//Manage data for read-only in PLC
stRoomDataPLC.bPirActive			:= stPirSensorData.bPrc;
stRoomDataPLC.uiActLuxLevel			:= TO_UINT(TRUNC(stPirSensorData.fBrightness));
stRoomDataPLC.uiActLightLevelPct	:= TO_UINT(TRUNC(arrfbLysGruppe[1].fbBallast.fActlLgtLvl_Prim));
		//stRoomDataPLC.uiActLightLevelPct	:= TO_UINT(TRUNC(fbLys.fbBallast.fActlLgtLvl_Prim)); //if only one group light control
stRoomDataPLC.uiBallastOnHours		:= uiBallastOnHours_MB; //The calculation for BallastOnHours is stored directly to the MB register below


//Assign data for read-only to MB registers
bPirActive_MB		:= stRoomDataPLC.bPirActive;
uiActLuxLevel_MB	:= stRoomDataPLC.uiActLuxLevel;

	//calculate BallastOnHours
	fbBallastOnHours(
		bEnableHourCount	:= bEnableHourCount,
		bPauseCount			:= arrfbLysGruppe[1].fbLightCtrl.bOffZone1,
		uiOnHours			:= uiBallastOnHours_MB,			//OnHours is updated here
		byOverflowCount		:= byOnHoursOverflowCount);


//Manage data for read/write for both PLC and MB registers
fbWriteSPLuxLevel(	nMaxValOut	:= uiMaxLuxLevel,
					nValIn1		:= uiSPLuxLevel_MB,		//nValIn1 takes priotity in case of download or restart
					nValIn2		:= stRoomDataPLC.uiSpLuxLevel,
					nValOut		=> uiLuxOn
				);


fbWritePirDelayTIme(	nMaxValOut	:= uiMaxPirOffMinutes,
						nValIn1		:= uiPirOffDelayTime_MB,		//nValIn1 takes priotity in case of download or restart
						nValIn2		:= stRoomDataPLC.uiPirOffDelayTime,
						nValOut		=> uiPirOffMinutes
					);
					

//Convert read/write modbus data to appropriate datatypes in PLC
fLuxOn	:= TO_REAL(uiLuxOn);			
tPIROff	:= TO_TIME(uiPirOffMinutes*udTimeScaling); //Time conversion defaults to ms

fLuxDim	:= TO_REAL(stRoomDataPLC.uiSpDimLuxLevel);			
tPIRDim	:= TO_TIME(stRoomDataPLC.uiPirDimDelayTime*udTimeScaling); //Time conversion defaults to ms
END_ACTION

ACTION A_Sensor:

fbSensor.ipCommunication := P_DALI_Background.arrfbKL6821Communication[Sensor_DALI_LINE_NUM];

//only 1 sensor
	
(*
fbSensor(
	byShrtAdr:= bySensorAddr,
	bInitialize:= bInitialize, 
	DALI_LINE_NUM:= Sensor_DALI_LINE_NUM, 
 	//bCancelHoldTimerOccupancy:= bCancelHoldTimerOccupancy, 
	stSensorSetup := stDaliSensorSetup,
	bInitErr=> bInitErr, 
	bInitDone=> bInitDone,
	stPirSensorData:= stPirSensorData, 
	arrSensorScales:= arrSensorScales);

*)
//several sensors	
fbSensor(
	arrShrtAdr:= arrSensorAddr,
	bInitialize:= bInitialize, 
	DALI_LINE_NUM:= Sensor_DALI_LINE_NUM, 
 	//bCancelHoldTimerOccupancy:= bCancelHoldTimerOccupancy, 
	stSensorSetup := stDaliSensorSetup,
	arrInitErr=> arrInitErr, 
	arrInitDone=> arrInitDone,
	stPirSensorData:= P_Foldedoer_4_517_Og_4_521_2Pcs.arrstPirSensorData_SepRoom[1], 
	arrSensorScales:= arrSensorScales);
	
	stPirSensorData := P_Foldedoer_4_517_Og_4_521_2Pcs.arrstPirSensorData_SepRoom[1]; //For at holde navngivning i ModbusComm
END_ACTION

END_PROGRAM

// ---- POUs/Alle_Rum/Rum_Med_DALI_Pir/Rum_4_513_Og_4_517_Og_4_521_Foldedoer/P_Rum_4_517.TcPOU
PROGRAM P_Rum_4_517
VAR

	arrfbLysGruppe			: ARRAY [1..2] OF FB_Light_Type_A;
	arrstDaliSetupGruppe	: ARRAY[1..2] OF SH_Light.ST_DALI_RoomSetup := 
	
													[(	byShrtAdr_Prim := 32, 
														byGrpAdr_Prim := 5, 
														eMod_Prim := E_DALIAddressType.Group, 
														//byShrtAdr_Sec := 1, 
														//byGrpAdr_Sec := 1, 
														//eMod_Sec := E_DALIAddressType.Short, 
														//byShrtAdr_Supl := 1,
														//eMod_Supl := E_DALIADDRESSTYPE.Group,
                                                        //byGrpAdr_Supl := 0, 
														DALI_LINE_NUM_PRIM := arrDALI_LINE_NUM_LIGHT[1], 
														DALI_LINE_NUM_SEC := 0, //0 = ingen zonestyring/vinduerække
														DALI_LINE_NUM_SUPL := arrDALI_LINE_NUM_PENDANTS[1]),
														
													(	byShrtAdr_Prim := 32, 
														byGrpAdr_Prim := 5, 
														eMod_Prim := E_DALIAddressType.Group, 
														//byShrtAdr_Sec := 1, 
														//byGrpAdr_Sec := 1, 
														//eMod_Sec := E_DALIAddressType.Short, 
														//byShrtAdr_Supl := 1, 
														DALI_LINE_NUM_PRIM := arrDALI_LINE_NUM_LIGHT[2], 
														DALI_LINE_NUM_SEC := 0, 
														DALI_LINE_NUM_SUPL := arrDALI_LINE_NUM_PENDANTS[2])];
														
	arrstLiveDataGruppe		: ARRAY [1..2] OF SH_Light.ST_LiveData;
	//stLiveData AT %MB22	: SH_Light.ST_LiveData;
	
	arrRunTuningGruppe: ARRAY[1..2] OF BOOL;
	
	
	
	bTopButtonZone1			: BOOL;
	bTopButtonZone1_Visu	: BOOL;
	bBottomButtonZone1		: BOOL;
	bBottomButtonZone1_Visu	: BOOL;
	bButtonZone2			: BOOL;
	bNeighborRoomsPir		: BOOL;
	fLuxOn					: REAL; 
	fLuxDim					: REAL;
	tPIRDim					: TIME;
	tPIROff					: TIME;
	fOffsetSec				: REAL := 20;
    bOccupiedRoom		    : BOOL;;
//Digital In
//    bDigitalPir AT %I*      : BOOL ;    

// Sensor Settings
	//fbSensor					: SH_Light.FB_NIKO_P46xx_1Pcs;
	fbSensor					: SH_Light.FB_NIKO_P46xx_2Pcs;
	//bySensorAddr				: BYTE := 9;
	arrSensorAddr				: ARRAY[1..2] OF BYTE := [3,4];
	bInitialize					: BOOL := TRUE;
	stDaliSensorSetup			: ST_DALI_NIKOP46SetupData := (
																nSensitivityPIRSegmentA := arrSensitivityOccupancy[1],
																nSensitivityPIRSegmentB := arrSensitivityOccupancy[2],
																nSensitivityPIRSegmentC := arrSensitivityOccupancy[3]);
	//bInitErr					: BOOL;
	//bInitDone					: BOOL;
	arrInitErr					: ARRAY [1..2] OF BOOL;
    arrInitDone					: ARRAY [1..2] OF BOOL;
	arrSensorScales				: ARRAY [1..10] OF SH_Light.ST_DALI_SensorScaleMode := [
																							(fMeassureMaxSensor := fMeassure_Zone5, fReadMaxSensor := fRead_Zone5),		
                                                                                            (fMeassureMaxSensor := fMeassure_Zone5, fReadMaxSensor := fRead_Zone5),																
																							8(())];
	bCancelHoldTimerOccupancy	: BOOL;
(*	eEventPriorityOccupancy		: E_DALIEventPriority := E_DALIEVENTPRIORITY.Middle;
	nHoldTimerOccupancy			: WORD := 5; // Value in s. 	
	nReportTimerOccupancy		: BYTE := 120; // Value in s, Preset manufacturer value
	nDeadtimeTimerOccupancy		: WORD := 100; // Value in ms, Predefined Value of DALI Standard
	bCancelHoldTimerOccupancy	: BOOL;
	nSensitivityOccupancy		: BYTE:= 3; //setting Sensivity (0..4) 0 (Off), 1 (Min), 2(Low), 3(High) and 4 (Max)

	bEnableLuxEvent				: BOOL;
	eEventPriorityBrightness	: E_DALIEventPriority := E_DALIEVENTPRIORITY.Middle;
	nDeadtimeTimerBrightness	: WORD := 1500; // Value in ms, Predefined Value of DALI Standard
	nHysteresisBrightness		: BYTE := 2; // Value in %
	nHysteresisMinBrightness	: BYTE := 10; // Absolute Value, depending on the manufacturer specific resolution
	nReportTimerBrightness		: BYTE := 120; // Value in s, Preset manufacturer value
*)


//ModbusComm setup
	
	fbWriteSPLuxLevel			: SH_Light.FB_TwoVal_SelectOne_RTrigChange;
	fbWritePirDelayTIme			: SH_Light.FB_TwoVal_SelectOne_RTrigChange;
	stRoomDataPLC				: SH_Light.ST_RoomDataPLC	:=	(	uiPirOffDelayTime	:= 30,
																	uiSpLuxLevel		:= 500,
																	uiPirDimDelayTime	:= 15,
																	uiSpDimLuxLevel		:= 200
																);
	fbBallastOnHours			: SH_Light.FB_CountOnHours;
	bEnableHourCount			: BOOL := TRUE;
	
	//Non-persistent modbus data
	bPirActive_MB			AT%MX562.0	: BOOL;				//bPirLys i gammel kode
	uiActLuxLevel_MB		AT%MB566	    : UINT;				//intHMIAktueltLux i gammel kode
	uiActLightLevelPct_MB	AT%MB570     : UINT;				//intDALI_Gruppe1_Lysniveau i gammel kode
	
	//For Conversion
	uiPirOffMinutes						: UINT;
	udTimeScaling						: UDINT := 60000;
	uiLuxOn								: UINT;
	
	//max values checks
	uiMaxLuxLevel						: UINT := 1023;
	uiMaxPirOffMinutes					: UINT := 180;
	
END_VAR

VAR CONSTANT
	Sensor_DALI_LINE_NUM: BYTE := 2;
	arrDALI_LINE_NUM_LIGHT: ARRAY[1..2] OF BYTE := [1,2]; //korrekt rækkefølge nødvendig //rækkefølge og linje 
	arrDALI_LINE_NUM_PENDANTS: ARRAY[1..2] OF BYTE := [0,0]; //korrekt rækkefølge nødvendig. 0 = ingen pendler
	arrSensitivityOccupancy				: ARRAY[1..3] OF BYTE := [4,4,4];
END_VAR
VAR PERSISTENT
	stPirSensorData: SH_Light.ST_DALI_Sensor;
	arrstTuneDataGruppe: ARRAY [1..2] OF SH_Light.ST_TuneData_EX;

	uiPirOffDelayTime_MB	AT%MB564	    : UINT;				//intHMI_Pir_SetValue i gammel kode
	uiSPLuxLevel_MB		    AT%MB568     : UINT;				//intHMI_Lux_SetValue i gammel kode
	uiBallastOnHours_MB	    AT%MB572	    : UINT;				//dintHMILysbraendtimer1 i gammel kode
	byOnHoursOverflowCount			    : BYTE;
END_VAR

///////)

A_Buttons();
A_LightCtrl();
A_ModbusComm();
A_Sensor();

ACTION A_Buttons:
(*
bTopButtonZone1		:= GVL_EnOcean.strEnOceanSwitch_Rum_4_517.bT1_ON OR bTopButtonZone1_Visu;
bBottomButtonZone1	:= GVL_EnOcean.strEnOceanSwitch_Rum_4_517.bT1_OFF OR bBottomButtonZone1_Visu;
*)

bTopButtonZone1		:= P_Foldedoer_4_517_Og_4_521_2Pcs.arrTopButtonZone1_ConnRoom[2] OR bTopButtonZone1_Visu;
bBottomButtonZone1	:= P_Foldedoer_4_517_Og_4_521_2Pcs.arrBottomButtonZone1_ConnRoom[2] OR bBottomButtonZone1_Visu;
END_ACTION

ACTION A_LightCtrl:

//gruppe 6
arrfbLysGruppe[1]( 
	nZoneID:= 1, 
	bButtonZone1:= bTopButtonZone1,
	bBottomButtonZone1 := bBottomButtonZone1,
	bTopButtonOverride := P_Foldedoer_4_517_Og_4_521_2Pcs.arrOverride_ConnRoom[2],
	//bButtonZone2:= bButtonZone2,
	fLuxOn:= fLuxOn, 
	fLuxDim:= fLuxDim, 
	tPIRDim:= tPIRDim, 
	tPIROff:= tPIROff, 
	fOffsetSec:= fOffsetSec, 
	bReInit:= , 
	stDaliSetup:= arrstDaliSetupGruppe[1], 
	ipCommunication_Prim:= P_DALI_Background.arrfbKL6821Communication[arrDALI_LINE_NUM_LIGHT[1]], 
	//ipCommunication_Sec:= P_DALI_Background.arrfbKL6821Communication[arrDALI_LINE_NUM_LIGHT[1]], //samme som lyslinjen, hvis den ikke eksisterer
	//ipCommunication_Supl:= P_DALI_Background.arrfbKL6821Communication[arrDALI_LINE_NUM_LIGHT[1]],//samme som lyslinjen, hvis den ikke eksisterer 
	fMinOutputPowerLevelRoom:= 15, 
	fMaxOutputPowerLevelRoom:= 100, 
	nCycleTimeInMS:= SH_Light.DALI_Param.nPlcTaskCycleTimeInMS*nDimCmdCycleTimeFactor,  //Used only for dim. Factor=2 makes dimming smooth
	bRunTuning:= arrRunTuningGruppe[1], 
	bOccupiedRoom=> , 
	bError_Prim=> , 
	nError_Prim=> , 
	stTuneData:=arrstTuneDataGruppe[1] , 
	stPirSensorData:= P_Foldedoer_4_517_Og_4_521_2Pcs.arrstPirSensorData_ConnRoom[2], 					//samme sensordata
	stLiveData:= arrstLiveDataGruppe[1]);


//gruppe 15	
arrfbLysGruppe[2]( 
	nZoneID:= 1, 
	bButtonZone1:= bTopButtonZone1,
	bBottomButtonZone1 := bBottomButtonZone1,
	bTopButtonOverride := P_Foldedoer_4_517_Og_4_521_2Pcs.arrOverride_ConnRoom[2],
	//bButtonZone2:= bButtonZone2,
	fLuxOn:= fLuxOn, 
	fLuxDim:= fLuxDim, 
	tPIRDim:= tPIRDim, 
	tPIROff:= tPIROff, 
	fOffsetSec:= fOffsetSec, 
	bReInit:= , 
	stDaliSetup:= arrstDaliSetupGruppe[2], 
	ipCommunication_Prim:= P_DALI_Background.arrfbKL6821Communication[arrDALI_LINE_NUM_LIGHT[2]], 
	//ipCommunication_Sec:= P_DALI_Background.arrfbKL6821Communication[arrDALI_LINE_NUM_LIGHT[2]], //samme som lyslinjen, hvis den ikke eksisterer
	//ipCommunication_Supl:= P_DALI_Background.arrfbKL6821Communication[arrDALI_LINE_NUM_LIGHT[2]], //samme som lyslinjen, hvis den ikke eksisterer 
	fMinOutputPowerLevelRoom:= 15, 
	fMaxOutputPowerLevelRoom:= 100, 
	nCycleTimeInMS:= SH_Light.DALI_Param.nPlcTaskCycleTimeInMS*nDimCmdCycleTimeFactor,  //Used only for dim. Factor=2 makes dimming smooth
	bRunTuning:= arrRunTuningGruppe[2], 
	bOccupiedRoom=> , 
	bError_Prim=> , 
	nError_Prim=> , 
	stTuneData:=arrstTuneDataGruppe[2] , 
	stPirSensorData:= P_Foldedoer_4_517_Og_4_521_2Pcs.arrstPirSensorData_ConnRoom[2], 					//samme sensordata
	stLiveData:= arrstLiveDataGruppe[2]);
END_ACTION

ACTION A_ModbusComm:
//Manage data for modbus communication

//Manage data for read-only in PLC
stRoomDataPLC.bPirActive			:= stPirSensorData.bPrc;
stRoomDataPLC.uiActLuxLevel			:= TO_UINT(TRUNC(stPirSensorData.fBrightness));
stRoomDataPLC.uiActLightLevelPct	:= TO_UINT(TRUNC(arrfbLysGruppe[1].fbBallast.fActlLgtLvl_Prim));
		//stRoomDataPLC.uiActLightLevelPct	:= TO_UINT(TRUNC(fbLys.fbBallast.fActlLgtLvl_Prim)); //if only one group light control
stRoomDataPLC.uiBallastOnHours		:= uiBallastOnHours_MB; //The calculation for BallastOnHours is stored directly to the MB register below


//Assign data for read-only to MB registers
bPirActive_MB		:= stRoomDataPLC.bPirActive;
uiActLuxLevel_MB	:= stRoomDataPLC.uiActLuxLevel;

	//calculate BallastOnHours
	fbBallastOnHours(
		bEnableHourCount	:= bEnableHourCount,
		bPauseCount			:= arrfbLysGruppe[1].fbLightCtrl.bOffZone1,
		uiOnHours			:= uiBallastOnHours_MB,			//OnHours is updated here
		byOverflowCount		:= byOnHoursOverflowCount);


//Manage data for read/write for both PLC and MB registers
fbWriteSPLuxLevel(	nMaxValOut	:= uiMaxLuxLevel,
					nValIn1		:= uiSPLuxLevel_MB,		//nValIn1 takes priotity in case of download or restart
					nValIn2		:= stRoomDataPLC.uiSpLuxLevel,
					nValOut		=> uiLuxOn
				);


fbWritePirDelayTIme(	nMaxValOut	:= uiMaxPirOffMinutes,
						nValIn1		:= uiPirOffDelayTime_MB,		//nValIn1 takes priotity in case of download or restart
						nValIn2		:= stRoomDataPLC.uiPirOffDelayTime,
						nValOut		=> uiPirOffMinutes
					);
					

//Convert read/write modbus data to appropriate datatypes in PLC
fLuxOn	:= TO_REAL(uiLuxOn);			
tPIROff	:= TO_TIME(uiPirOffMinutes*udTimeScaling); //Time conversion defaults to ms

fLuxDim	:= TO_REAL(stRoomDataPLC.uiSpDimLuxLevel);			
tPIRDim	:= TO_TIME(stRoomDataPLC.uiPirDimDelayTime*udTimeScaling); //Time conversion defaults to ms
END_ACTION

ACTION A_Sensor:

fbSensor.ipCommunication := P_DALI_Background.arrfbKL6821Communication[Sensor_DALI_LINE_NUM];

//only 1 sensor
	
(*
fbSensor(
	byShrtAdr:= bySensorAddr,
	bInitialize:= bInitialize, 
	DALI_LINE_NUM:= Sensor_DALI_LINE_NUM, 
 	//bCancelHoldTimerOccupancy:= bCancelHoldTimerOccupancy, 
	stSensorSetup := stDaliSensorSetup,
	bInitErr=> bInitErr, 
	bInitDone=> bInitDone,
	stPirSensorData:= stPirSensorData, 
	arrSensorScales:= arrSensorScales);

*)
//several sensors	
fbSensor(
	arrShrtAdr:= arrSensorAddr,
	bInitialize:= bInitialize, 
	DALI_LINE_NUM:= Sensor_DALI_LINE_NUM, 
 	//bCancelHoldTimerOccupancy:= bCancelHoldTimerOccupancy, 
	stSensorSetup := stDaliSensorSetup,
	arrInitErr=> arrInitErr, 
	arrInitDone=> arrInitDone,
	stPirSensorData:= P_Foldedoer_4_517_Og_4_521_2Pcs.arrstPirSensorData_SepRoom[2],
	arrSensorScales:= arrSensorScales);
	
	stPirSensorData := P_Foldedoer_4_517_Og_4_521_2Pcs.arrstPirSensorData_SepRoom[2]; //For at holde navngivning i ModbusComm
END_ACTION

END_PROGRAM

// ---- POUs/DALI/DALI_Setup/FBs/FB_Part102Scenes.TcPOU
FUNCTION_BLOCK FB_Part102Scenes
VAR_INPUT
	ipDALICommunication		:	I_DALICommunication;
END_VAR
VAR_OUTPUT
	bBusy					:	BOOL;
END_VAR
VAR
	{region "Visu"}
	nScene					:	BYTE;
	bGoToScene				:	BOOL;
	bSwitchOff				:	BOOL;
	bRead					:	BOOL;
	bWrite		 			:	BOOL;
	aScene					:	ARRAY [0..63] OF BYTE;
	aNoShortAddress			:	ARRAY [0..63] OF BOOL;
	bHideWaitSymbol			:	BOOL := TRUE;
	{endregion}
	nStep					:	INT; // Running index
	nAddress				:	INT;
	aFont					:	ARRAY [0..63] OF DWORD;

	fb103StartQuiescentMode	:	FB_DALI103StartQuiescentMode(0);
	fb103StopQuiescentMode	:	FB_DALI103StopQuiescentMode(0);
	fb102QuerySceneLevel	:	FB_DALI102QuerySceneLevel(0);
	fb102SetScene			:	FB_DALI102SetScene(0);
	fb102GoToScene			:	FB_DALI102GoToScene(0);
	fb102Off				:	FB_DALI102Off(0);
END_VAR

{region "Detect Commands"}
IF (bRead AND (nStep = 0)) THEN 
	nStep := 5;
	bRead := FALSE;
	bHideWaitSymbol := FALSE;
END_IF

IF (bWrite AND (nStep = 0)) THEN 
	nStep := 20;
	bWrite := FALSE;
	bHideWaitSymbol := FALSE;
END_IF

IF (bGoToScene AND (nStep = 0)) THEN 
	nStep := 30;
	bGoToScene := FALSE;
	bHideWaitSymbol := FALSE;
END_IF

IF (bSwitchOff AND (nStep = 0)) THEN
	nStep := 40;
	bSwitchOff := FALSE;
	bHideWaitSymbol := FALSE;
END_IF
{endregion}
{region "Manage Dialog Selection}
IF (nStep = 0) THEN
	bBusy := FALSE;
ELSE
	bBusy := TRUE;
END_IF
{endregion}
{region "Execute Commands"}
CASE nStep OF
0:
{region "Init"}
	bRead := FALSE;	
	bWrite := FALSE;
	bGoToScene := FALSE;
	bSwitchOff := FALSE;
	bHideWaitSymbol := TRUE;
	nAddress := 0;

	fb103StartQuiescentMode.ipDALICommunication := ipDALICommunication;
	fb103StopQuiescentMode.ipDALICommunication := ipDALICommunication;
	fb102QuerySceneLevel.ipDALICommunication := ipDALICommunication;
	fb102SetScene.ipDALICommunication := ipDALICommunication;
	fb102GoToScene.ipDALICommunication := ipDALICommunication;
	fb102Off.ipDALICommunication := ipDALICommunication;
{endregion}
5:
{region "Start Qiescent Mode"}
	fb103StartQuiescentMode(bStart := TRUE,
							eAddressType := Tc3_DALI.E_DALIAddressType.Broadcast,
							eCommandPriority := Tc3_DALI.E_DALICommandPriority.Middle);
	IF (NOT fb103StartQuiescentMode.bBusy) THEN
		fb103StartQuiescentMode(bStart:= FALSE);
		nStep := 10;
	END_IF
{endregion}
10:
{region "Query Scene Level"}
	fb102QuerySceneLevel(	bStart := TRUE,
							nAddress := TO_BYTE(nAddress),
							eAddressType := Tc3_DALI.E_DALIAddressType.Short,
							eCommandPriority := Tc3_DALI.E_DALICommandPriority.Middle,
							nScene := nScene,
							nSceneLevel=> aScene[nAddress]);
	IF (NOT fb102QuerySceneLevel.bBusy) THEN
		fb102QuerySceneLevel (bStart:= FALSE);
		IF (fb102QuerySceneLevel.ipResultMessage.nEventId = TC_EVENTS.TcDALIEventClass.NoResponseFromTheDALIDevice.nEventId) THEN // Deletes not existing short addresses from display
			aNoShortAddress[nAddress] := TRUE;
			aFont[nAddress] := 16#FF505050;
		ELSE
			aNoShortAddress[nAddress] := FALSE;
			aFont[nAddress] := 16#FFFFFFFF;
		END_IF
		nAddress := nAddress + 1;
		IF (nAddress > 63)THEN
			nStep := 15;
		END_IF
	END_IF
{endregion}
15:
{region "Stop Qiescent Mode"}
	fb103StopQuiescentMode(	bStart := TRUE,
							eAddressType := Tc3_DALI.E_DALIAddressType.Broadcast,
							eCommandPriority := Tc3_DALI.E_DALICommandPriority.Middle);
	IF (NOT fb103StopQuiescentMode.bBusy) THEN
		fb103StopQuiescentMode(	bStart:= FALSE);
		nStep := 0;
	END_IF
{endregion}
20:
{region "Set Scene"}
	IF (aNoShortAddress[nAddress] = TRUE) THEN
		nAddress := nAddress + 1;
		IF (nAddress > 63)THEN
			nStep := 0;
		END_IF
	ELSE
		fb102SetScene(	bStart := TRUE,
						nAddress := TO_BYTE(nAddress),
						eAddressType := Tc3_DALI.E_DALIAddressType.Short,
						eCommandPriority := Tc3_DALI.E_DALICommandPriority.Middle,
						nSceneLevel := aScene[nAddress],
						nScene := nScene);
		IF (NOT fb102SetScene.bBusy) THEN
			fb102SetScene(bStart := FALSE);
			nAddress := nAddress + 1;
			IF (nAddress > 63)THEN
				nStep := 0;
			END_IF
		END_IF
	END_IF
{endregion}
30:
{region "Go To Scene"}
	IF (aNoShortAddress[nAddress] = TRUE) THEN
		nAddress := nAddress + 1;
		IF (nAddress > 63)THEN
			nStep := 0;
		END_IF
	ELSE
		fb102GoToScene(	bStart := TRUE,
						nAddress := TO_BYTE(nAddress),
						eAddressType := Tc3_DALI.E_DALIAddressType.Short,
						eCommandPriority := Tc3_DALI.E_DALICommandPriority.Middle,
						nScene := nScene);
		IF (NOT fb102GoToScene.bBusy) THEN
			fb102GoToScene(bStart := FALSE);
			nAddress := nAddress + 1;
			IF (nAddress > 63)THEN
				nStep := 0;
			END_IF
		END_IF
	END_IF
{endregion}
40:
{region "Switch Off"}
	fb102Off(	bStart := TRUE,
				nAddress := TO_BYTE(nAddress),
				eAddressType := Tc3_DALI.E_DALIAddressType.Broadcast,
				eCommandPriority := Tc3_DALI.E_DALICommandPriority.Middle);
	IF (NOT fb102Off.bBusy) THEN
		fb102Off(bStart := FALSE);
		nStep := 0;
	END_IF
{endregion}
END_CASE
{endregion}

END_FUNCTION_BLOCK

// ---- POUs/DALI/DALI_Setup/FBs/FB_Part300GenericDevice.TcPOU
FUNCTION_BLOCK FB_Part300GenericDevice
VAR_INPUT
	ipDALICommunication			:	I_DALICommunication;
END_VAR
VAR_OUTPUT
	bBusy						:	BOOL;
END_VAR
VAR
	{region "Visu"}
	nInputValue					:	LWORD;
	nInstanceError				:	BYTE;
	nResolution					:	BYTE;
	eEventScheme				:	E_DALIEventScheme;
	nEventFilter				:	DWORD;
	bRead						:	BOOL;
	bWrite						:	BOOL;
	bEnable						:	BOOL;
	bBit0						:	BOOL;
	bBit1						:	BOOL;
	bBit2						:	BOOL;
	bBit3						:	BOOL;
	bBit4						:	BOOL;
	bBit5						:	BOOL;
	bBit6						:	BOOL;
	bBit7						:	BOOL;
	eEventPriority				:	E_DALIEventPriority := E_DALIEventPriority.Middle;
	{endregion}
	nStep						:	INT;
	nAddress					:	BYTE;
	nInstanceAddress			:	BYTE;
	bHideWaitSymbol				:	BOOL := TRUE;

	fb103StartQuiescentMode		:	FB_DALI103StartQuiescentMode(0);
	fb103StopQuiescentMode		:	FB_DALI103StopQuiescentMode(0);
	fb103QueryInstanceError		:	FB_DALI103QueryInstanceError(0);
	fb103QueryInstanceStatus	:	FB_DALI103QueryInstanceStatus(0);
	fb103QueryResolution		:	FB_DALI103QueryResolution(0);
	fb103QueryInputValue 		:	FB_DALI103QueryInputValue(0);
	fb103QueryEventScheme 		:	FB_DALI103QueryEventScheme(0);
	fb103QueryEventFilter 		:	FB_DALI103QueryEventFilter(0);
	fb103QueryEventPriority		:	FB_DALI103QueryEventPriority(0);
	fb103EnableInstance 		:	FB_DALI103EnableInstance(0);
	fb103DisableInstance		:	FB_DALI103DisableInstance(0);
	fb103SetEventScheme 		:	FB_DALI103SetEventScheme(0);
	fb103SetEventFilter 		:	FB_DALI103SetEventFilter(0);
	fb103SetEventPriority		:	FB_DALI103SetEventPriority(0);
END_VAR

{region "Detect Commands"}
IF (bRead AND (nStep = 0)) THEN
	nStep := 5;
	bRead := FALSE;
	bHideWaitSymbol := FALSE;
END_IF

IF (bWrite AND (nStep = 0)) THEN
	nStep := 1000;
	bWrite := FALSE;
	bHideWaitSymbol := FALSE;
END_IF
{endregion}
{region "Manage Dialog Selection}
IF (nStep = 0) THEN
	bBusy := FALSE;
ELSE
	bBusy := TRUE;
END_IF
{endregion}
{region "Execute Commands"}
CASE nStep OF
0:
{region "Init"}
	bRead := FALSE;
	bWrite := FALSE;
	bHideWaitSymbol := TRUE;

	fb103StartQuiescentMode.ipDALICommunication := ipDALICommunication;
	fb103StopQuiescentMode.ipDALICommunication := ipDALICommunication;
	fb103QueryInstanceError.ipDALICommunication := ipDALICommunication;
	fb103QueryInstanceStatus.ipDALICommunication := ipDALICommunication;
	fb103QueryResolution.ipDALICommunication := ipDALICommunication;
	fb103QueryInputValue.ipDALICommunication := ipDALICommunication;
	fb103QueryEventScheme.ipDALICommunication := ipDALICommunication;
	fb103QueryEventFilter.ipDALICommunication := ipDALICommunication;
	fb103QueryEventPriority.ipDALICommunication := ipDALICommunication;
	fb103EnableInstance.ipDALICommunication := ipDALICommunication;
	fb103DisableInstance.ipDALICommunication := ipDALICommunication;
	fb103SetEventScheme.ipDALICommunication := ipDALICommunication;
	fb103SetEventFilter.ipDALICommunication := ipDALICommunication;
	fb103SetEventPriority.ipDALICommunication := ipDALICommunication;
{endregion}
{region "Read"}
5:
{region "Start Qiescent Mode"}
	fb103StartQuiescentMode(bStart := TRUE,
							eAddressType := Tc3_DALI.E_DALIAddressType.Broadcast,
							eCommandPriority := Tc3_DALI.E_DALICommandPriority.Middle);
	IF (NOT fb103StartQuiescentMode.bBusy) THEN
		fb103StartQuiescentMode(bStart:= FALSE);
		nStep := 10;
	END_IF
{endregion}
10:
{region "Query Instance Error"}
	fb103QueryInstanceError(bStart := TRUE,
							nAddress := nAddress,
							eAddressType := Tc3_DALI.E_DALIAddressType.Short,
							nInstanceAddress := nInstanceAddress,
							eInstanceAddressType := Tc3_DALI.E_DALIInstanceAddressType.InstanceNumber,
							eCommandPriority := Tc3_DALI.E_DALICommandPriority.Middle,
							nInstanceError=> nInstanceError);
	IF (NOT fb103QueryInstanceError.bBusy) THEN
		fb103QueryInstanceError(bStart := FALSE);
		nStep := 20;
	END_IF
{endregion}
20:
{region "Query Instance Status"}
	fb103QueryInstanceStatus(	bStart := TRUE,
								nAddress := nAddress,
								eAddressType := Tc3_DALI.E_DALIAddressType.Short,
								nInstanceAddress := nInstanceAddress,
								eInstanceAddressType := Tc3_DALI.E_DALIInstanceAddressType.InstanceNumber,
								eCommandPriority := Tc3_DALI.E_DALICommandPriority.Middle);
	IF (NOT fb103QueryInstanceStatus.bBusy) THEN
		fb103QueryInstanceStatus(bStart := FALSE);
		IF (fb103QueryInstanceStatus.nInstanceStatus.1) THEN
			bEnable := TRUE;
		END_IF
		nStep := 30;
	END_IF
30:
{region "Query Resolution"}
	fb103QueryResolution(	bStart := TRUE,
							nAddress := nAddress,
							eAddressType := Tc3_DALI.E_DALIAddressType.Short,
							nInstanceAddress := nInstanceAddress,
							eInstanceAddressType := Tc3_DALI.E_DALIInstanceAddressType.InstanceNumber,
							eCommandPriority := Tc3_DALI.E_DALICommandPriority.Middle,
							nResolution => nResolution);
	IF (NOT fb103QueryResolution.bBusy) THEN
		fb103QueryResolution(bStart := FALSE);
		nStep := 40;
	END_IF
{endregion}
40:
{region "Query Input Value"}
	fb103QueryInputValue(	bStart := TRUE,
							nAddress := nAddress,
							eAddressType := Tc3_DALI.E_DALIAddressType.Short,
							nInstanceAddress := nInstanceAddress,
							eInstanceAddressType := Tc3_DALI.E_DALIInstanceAddressType.InstanceNumber,
							eCommandPriority := Tc3_DALI.E_DALICommandPriority.Middle,
							nResolution := nResolution,
							nInputValue => nInputValue);
	IF (NOT fb103QueryInputValue.bBusy) THEN
		fb103QueryInputValue(bStart := FALSE);
		nStep := 50;
	END_IF
{endregion}
50:
{region "Query Event Scheme"}
	fb103QueryEventScheme(	bStart := TRUE,
							nAddress := nAddress,
							eAddressType := Tc3_DALI.E_DALIAddressType.Short,
							nInstanceAddress := nInstanceAddress,
							eInstanceAddressType := Tc3_DALI.E_DALIInstanceAddressType.InstanceNumber,
							eCommandPriority := Tc3_DALI.E_DALICommandPriority.Middle,
							eEventScheme => eEventScheme);
	IF (NOT fb103QueryEventScheme.bBusy) THEN
		fb103QueryEventScheme(bStart := FALSE);
		nStep := 60;
	END_IF
{endregion}
60:
{region "Query Event Filter"}
	fb103QueryEventFilter(	bStart := TRUE,
							nAddress := nAddress,
							eAddressType := Tc3_DALI.E_DALIAddressType.Short,
							nInstanceAddress := nInstanceAddress,
							eInstanceAddressType := Tc3_DALI.E_DALIInstanceAddressType.InstanceNumber,
							eCommandPriority := Tc3_DALI.E_DALICommandPriority.Middle,
							nEventFilter=> nEventFilter);
	IF (NOT fb103QueryEventFilter.bBusy) THEN
		fb103QueryEventFilter(bStart := FALSE);
		bBit0 := nEventFilter.0;
		bBit1 := nEventFilter.1;
		bBit2 := nEventFilter.2;
		bBit3 := nEventFilter.3;
		bBit4 := nEventFilter.4;
		bBit5 := nEventFilter.5;
		bBit6 := nEventFilter.6;
		bBit7 := nEventFilter.7;
		nStep := 90;
	END_IF
{endregion}
90:
{region "Query Event Priority"}
	fb103QueryEventPriority(bStart := TRUE,
							nAddress := nAddress,
							eAddressType := Tc3_DALI.E_DALIAddressType.Short,
							nInstanceAddress := nInstanceAddress,
							eInstanceAddressType := Tc3_DALI.E_DALIInstanceAddressType.InstanceNumber,
							eCommandPriority := Tc3_DALI.E_DALICommandPriority.Middle,
							eEventPriority=> eEventPriority);
	IF (NOT fb103QueryEventPriority.bBusy) THEN
		fb103QueryEventPriority(bStart := FALSE);
		nStep := 100;
	END_IF
{endregion}
100:
{region "Stop Qiescent Mode"}
	fb103StopQuiescentMode(	bStart := TRUE,
							eAddressType := Tc3_DALI.E_DALIAddressType.Broadcast,
							eCommandPriority := Tc3_DALI.E_DALICommandPriority.Middle);
	IF (NOT fb103StopQuiescentMode.bBusy) THEN
		fb103StopQuiescentMode(	bStart := FALSE);
		nStep := 0;
	END_IF
{endregion}
{endregion}

{region "Write"}
1000:	
{region "Enable or Disable Instance"}
	IF (bEnable) THEN
		fb103EnableInstance(bStart := TRUE,
							nAddress := nAddress,
							eAddressType := Tc3_DALI.E_DALIAddressType.Short,
							nInstanceAddress := nInstanceAddress,
							eInstanceAddressType := Tc3_DALI.E_DALIInstanceAddressType.InstanceNumber,
							eCommandPriority := Tc3_DALI.E_DALICommandPriority.Middle);
		IF (NOT fb103EnableInstance.bBusy) THEN
			fb103EnableInstance(bStart := FALSE);
			nStep := 1010;
		END_IF
	ELSE
		fb103DisableInstance(bStart := TRUE,
							 nAddress := nAddress,
							 eAddressType := Tc3_DALI.E_DALIAddressType.Short,
							 nInstanceAddress := nInstanceAddress,
							 eInstanceAddressType := Tc3_DALI.E_DALIInstanceAddressType.InstanceNumber,
							 eCommandPriority := Tc3_DALI.E_DALICommandPriority.Middle);
		IF (NOT fb103DisableInstance.bBusy) THEN
			fb103DisableInstance(bStart := FALSE);
			nStep := 0;
		END_IF
	END_IF
{endregion}
1010:
{region "Set Event Scheme"}
	fb103SetEventScheme(bStart := TRUE,
						nAddress := nAddress,
						eAddressType := Tc3_DALI.E_DALIAddressType.Short,
						nInstanceAddress := nInstanceAddress,
						eInstanceAddressType := Tc3_DALI.E_DALIInstanceAddressType.InstanceNumber,
						eCommandPriority := Tc3_DALI.E_DALICommandPriority.Middle,
						eEventScheme := eEventScheme);
	IF (NOT fb103SetEventScheme.bBusy) THEN
		fb103SetEventScheme(bStart := FALSE);
		nStep := 1020;
	END_IF
{endregion}
1020:
{region "Set Event Filter"}
	nEventFilter.0 := bBit0;
	nEventFilter.1 := bBit1;
	nEventFilter.2 := bBit2;
	nEventFilter.3 := bBit3;
	nEventFilter.4 := bBit4;
	nEventFilter.5 := bBit5;
	nEventFilter.6 := bBit6;
	nEventFilter.7 := bBit7;
	fb103SetEventFilter(bStart := TRUE,
						nAddress := nAddress,
						eAddressType := Tc3_DALI.E_DALIAddressType.Short,
						nInstanceAddress := nInstanceAddress,
						eInstanceAddressType := Tc3_DALI.E_DALIInstanceAddressType.InstanceNumber,
						eCommandPriority := Tc3_DALI.E_DALICommandPriority.Middle,
						nEventFilter := nEventFilter);
	IF (NOT fb103SetEventFilter.bBusy) THEN
		fb103SetEventFilter(bStart := FALSE);
		nStep := 1050;
	END_IF
{endregion}
1050:
{region "Set Event Priority"}
	fb103SetEventPriority(	bStart := TRUE,
							nAddress := nAddress,
							eAddressType := Tc3_DALI.E_DALIAddressType.Short,
							nInstanceAddress := nInstanceAddress,
							eInstanceAddressType := Tc3_DALI.E_DALIInstanceAddressType.InstanceNumber,
							eCommandPriority := Tc3_DALI.E_DALICommandPriority.Middle,
							eEventPriority:= eEventPriority);
	IF (NOT fb103SetEventPriority.bBusy) THEN
		fb103SetEventPriority(bStart := FALSE);
		nStep := 0;
	END_IF
{endregion}
{endregion}
END_CASE
{endregion}
{endregion}

END_FUNCTION_BLOCK

// ---- POUs/EnOcean/P_EnOcean.TcPOU
PROGRAM P_EnOcean
VAR
	fbKL6581			: FB_KL6581;
	stKL6581_in  AT %I* : KL6581_INPUT;
	stKL6581_out AT %Q*	: KL6581_OUTPUT;
	stKL6581			: STR_KL6581;
	bInitCom			: BOOL := TRUE;
	
	arrEnOcean_Search	: ARRAY [1..8] OF FB_EnOcean_Search;
	nSearchIdx			: BYTE;
	bSerach				: BOOL;
	arrDevices			: ARRAY [1..8] OF INT;
	arrID				: ARRAY [1..8, 0..255] OF DWORD;
	
		//Trykknapper Atrium
	fbAtriumNiveau_Tryk_PladeB				: FB_Rec_RPS_Switch;
	fbAtriumNiveau_Tryk_Sevice				: FB_Rec_RPS_Switch;			

	//Trykknapper på gange

	
	//Trykknapper i rum
	fbRum_4_513_Tryk_Indgang1_1						: FB_Rec_RPS_Switch;
	fbRum_4_513_Tryk_Indgang1_2						: FB_Rec_RPS_Switch;
	fbRum_4_513_Tryk_Indgang2						: FB_Rec_RPS_Switch;
    fbRum_4_517_Tryk                                : FB_Rec_RPS_Switch;
	fbRum_4_521_Tryk_Indgang1                       : FB_Rec_RPS_Switch;
    fbRum_4_521_Tryk_Indgang2                       : FB_Rec_RPS_Switch;
	fbGang_4_531_Tryk                               : FB_Rec_RPS_Switch;

END_VAR

VAR CONSTANT
	byNode_1: BYTE := 1;
	byNode_2: BYTE := 2;
	byNode_3: BYTE := 3;
	byNode_4: BYTE := 4;
	byNode_5: BYTE := 5;
	byNode_6: BYTE := 6;
	byNode_7: BYTE := 7;
	byNode_8: BYTE := 8;
END_VAR


(* Kommunikation mit der KL6581. *)
(* Communication with the KL6581. *)
fbKL6581(
	bInit			:= bInitCom,
	nIdx			:= 2,
	stKL6581_in		:= stKL6581_In,
	stKL6581_out	:= stKL6581_Out,
	bReady			=> ,
	bBusy			=> ,
	bError			=> ,
	iErrorID		=> ,
	str_KL6581		=> stKL6581);

GVL_AHDataModbus.EnOceanError	:= TO_UINT(fbKL6581.iErrorID);
(* Warten bis der Kommunikationsbaustein initialisiert wurde.*)
(* Wait until the communication function block has been initialized. *)
IF (NOT fbKL6581.bReady) THEN
	RETURN;
END_IF

FOR nSearchIdx:= 1 TO 8 DO
	arrEnOcean_Search[nSearchIdx](
		bStart:= TRUE, 
		str_KL6581:= stKL6581 , 
		byNode:= nSearchIdx, 
		bReceive=> , 
		iDevices=>arrDevices[nSearchIdx] , 
		ar_ID=> );
		
		MEMCPY(ADR(arrID[nSearchIdx,0]), ADR(arrEnOcean_Search[nSearchIdx].ar_ID), SIZEOF(arrEnOcean_Search[nSearchIdx].ar_ID)); 
END_FOR

//Gange



//RUM
 //
P_Rum_4_513();
P_Rum_4_517();
P_Rum_4_521();
P_Rum_4_531();


//AtriumNiveau
A_AtriumNiveau();

ACTION A_AtriumNiveau:
fbAtriumNiveau_Tryk_PladeB(
	str_KL6581:=stKL6581 , 
	byNode:=0, 
	dw_ID:= 16#0029B92D, 
	str_EnOceanSwitch=> GVL_EnOcean.strEnOceanSwitch_AtriumNiveau_PladeB,
	by_Node=> , 
	bReceive=> );

//knap 2 
(*
fbAtriumNiveau_Tryk_Sevice(
	str_KL6581:=stKL6581 , 
	byNode:=0, 
	dw_ID:= 16#00FEE4FE87, 
	str_EnOceanSwitch=> GVL_EnOcean.strEnOceanSwitch_AtriumNiveau_Service, 
	by_Node=> , 
	bReceive=> );
*)
END_ACTION

ACTION P_Rum_4_513:
fbRum_4_513_Tryk_Indgang1_1(
	str_KL6581:=stKL6581 , 
	byNode:=2 , 
	dw_ID:=  16#0029AB59, 
	str_EnOceanSwitch=> GVL_EnOcean.strEnOceanSwitch_Rum_4_513_Indgang1_1, 
	by_Node=> , 
	bReceive=> );
//bt1 
fbRum_4_513_Tryk_Indgang1_2(
	str_KL6581:=stKL6581 , 
	byNode:=2 , 
	dw_ID:=  16#002A4F50, 
	str_EnOceanSwitch=> GVL_EnOcean.strEnOceanSwitch_Rum_4_513_Indgang1_2, 
	by_Node=> , 
	bReceive=> );
	//bt2 Invers
fbRum_4_513_Tryk_Indgang2(
	str_KL6581:=stKL6581 , 
	byNode:=2 , 
	dw_ID:=  16#0029AB5B, 
	str_EnOceanSwitch=> GVL_EnOcean.strEnOceanSwitch_Rum_4_513_Indgang2, 
	by_Node=> , 
	bReceive=> );
	//BT1
END_ACTION

ACTION P_Rum_4_517:
fbRum_4_517_Tryk(
	str_KL6581:=stKL6581 , 
	byNode:=2 , 
	dw_ID:= 16#0029ABB8, 
	str_EnOceanSwitch=> GVL_EnOcean.strEnOceanSwitch_Rum_4_517, 
	by_Node=> , 
	bReceive=> );
//BT1
END_ACTION

ACTION P_Rum_4_521:
fbRum_4_521_Tryk_Indgang1(
	str_KL6581:=stKL6581 , 
	byNode:=2 , 
	dw_ID:= 16#0029ABB5, 
	str_EnOceanSwitch=> GVL_EnOcean.strEnOceanSwitch_Rum_4_521_Indgang1, 
	by_Node=> , 
	bReceive=> );
//BT1
	
fbRum_4_521_Tryk_Indgang2(
	str_KL6581:=stKL6581 , 
	byNode:=2 , 
	dw_ID:= 16#0029AB62, 
	str_EnOceanSwitch=> GVL_EnOcean.strEnOceanSwitch_Rum_4_521_Indgang2, 
	by_Node=> , 
	bReceive=> );
//BT2 Invers
END_ACTION

ACTION P_Rum_4_531:
fbGang_4_531_Tryk(
	str_KL6581:=stKL6581 , 
	byNode:=2 , 
	dw_ID:=  16#0029AB93, 
	str_EnOceanSwitch=> GVL_EnOcean.strEnOceanSwitch_Rum_4_531, 
	by_Node=> , 
	bReceive=> );
//bt2
END_ACTION

END_PROGRAM

// ---- POUs/Alle_Rum/Gange/Gang_7_501/Visualization_4_330_3.TcVIS
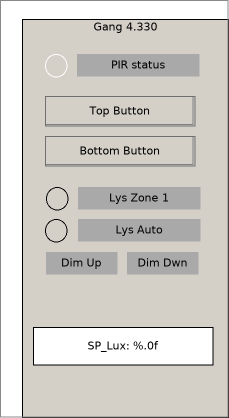
VISUALIZATION Visualization_4_330_3  // 229x418
    RoundedRectangle (22,19 207x399), "Gang 4.330"
    Rectangle (33,327 180x38), "SP_Lux: %.0f", text variable: P_Gang_2_143A.arrfbLysGruppe[1].fbLightCtrl.fLuxZone1
    Button (45,96 150x30), "Top Button"
        tap P_Gang_2_143A.bTopButtonZone1_Visu
    Button (45,136 150x30), "Bottom Button"
        tap P_Gang_2_143A.bBottomButtonZone1_Visu
    Ellipse (46,187 22x23), colour toggle: P_Gang_2_143A.fbLys.fbLightCtrl.bOnZone1
    Rectangle (78,187 122x22), "Lys Zone 1"
    Rectangle (46,252 71x22), "Dim Up", colour toggle: P_Gang_2_143A.arrfbLysGruppe[1].fbLightCtrl.bDimUp
    Rectangle (127,252 71x22), "Dim Dwn", colour toggle: P_Gang_2_143A.arrfbLysGruppe[1].fbLightCtrl.bDimDwn
    Ellipse (45,219 22x23), colour toggle: P_Gang_2_143A.arrfbLysGruppe[1].fbLightCtrl.bAutoZone1
    Rectangle (78,219 122x22), "Lys Auto"
    Ellipse (45,54 22x23), colour toggle: P_Gang_2_143A.arrfbLysGruppe[1].fbLightCtrl.bPIR
    Rectangle (77,54 122x22), "PIR status"
END_VISUALIZATION

// ---- POUs/Alle_Rum/Gange/Gang_4_531A/Visualization_5_338_1_1_1_1_2_1_1_1_1.TcVIS
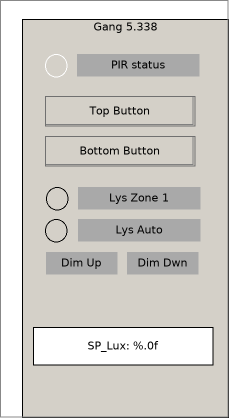
VISUALIZATION Visualization_5_338_1_1_1_1_2_1_1_1_1  // 229x418
    RoundedRectangle (22,19 207x399), "Gang 5.338"
    Rectangle (33,327 180x38), "SP_Lux: %.0f", text variable: P_Gang_5_338.arrfbLysGruppe[1].fbLightCtrl.fLuxZone1
    Button (45,96 150x30), "Top Button"
        tap P_Gang_5_338.bTopButtonZone1_Visu
    Button (45,136 150x30), "Bottom Button"
        tap P_Gang_5_338.bBottomButtonZone1_Visu
    Ellipse (46,187 22x23), colour toggle: P_Gang_5_338.arrfbLysGruppe[1].fbLightCtrl.bOnZone1
    Rectangle (78,187 122x22), "Lys Zone 1"
    Rectangle (46,252 71x22), "Dim Up", colour toggle: P_Gang_5_338.arrfbLysGruppe[1].fbLightCtrl.bDimUp
    Rectangle (127,252 71x22), "Dim Dwn", colour toggle: P_Gang_5_338.arrfbLysGruppe[1].fbLightCtrl.bDimDwn
    Ellipse (45,219 22x23), colour toggle: P_Gang_5_338.arrfbLysGruppe[1].fbLightCtrl.bAutoZone1
    Rectangle (78,219 122x22), "Lys Auto"
    Ellipse (45,54 22x23), colour toggle: P_Gang_5_338.arrfbLysGruppe[1].fbLightCtrl.bPIR
    Rectangle (77,54 122x22), "PIR status"
END_VISUALIZATION

// ---- POUs/Alle_Rum/Rum_Med_DALI_Pir/Rum_4_513_Og_4_517_Og_4_521_Foldedoer/Visualization_5_352_1_1_1_1_1_1_1.TcVIS
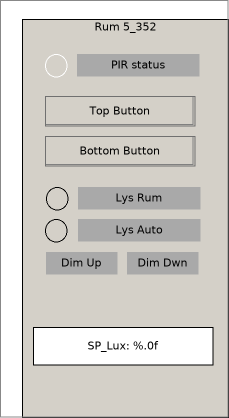
VISUALIZATION Visualization_5_352_1_1_1_1_1_1_1  // 229x418
    RoundedRectangle (22,19 207x399), "Rum 5_352"
    Rectangle (33,327 180x38), "SP_Lux: %.0f", text variable: P_Rum_4_324.fbLys.fbLightCtrl.fLuxZone1
    Button (45,96 150x30), "Top Button"
        tap P_Rum_5_352.bTopButtonZone1_Visu
    Button (45,136 150x30), "Bottom Button"
        tap P_Rum_5_352.bBottomButtonZone1_Visu
    Ellipse (46,187 22x23), colour toggle: P_Rum_5_352.fbLys.fbLightCtrl.bOnZone1
    Rectangle (78,187 122x22), "Lys Rum"
    Rectangle (46,252 71x22), "Dim Up", colour toggle: P_Rum_5_352.fbLys.fbLightCtrl.bDimUp
    Rectangle (127,252 71x22), "Dim Dwn", colour toggle: P_Rum_5_352.fbLys.fbLightCtrl.bDimDwn
    Ellipse (45,219 22x23), colour toggle: P_Rum_5_352.fbLys.fbLightCtrl.bAutoZone1
    Rectangle (78,219 122x22), "Lys Auto"
    Ellipse (45,54 22x23), colour toggle: P_Rum_5_352.fbLys.fbLightCtrl.bPIR
    Rectangle (77,54 122x22), "PIR status"
END_VISUALIZATION

// ---- POUs/DALI/DALI_Setup/VISUs/Visu_DALICommissioning/Visu_Part102Commands.TcVIS
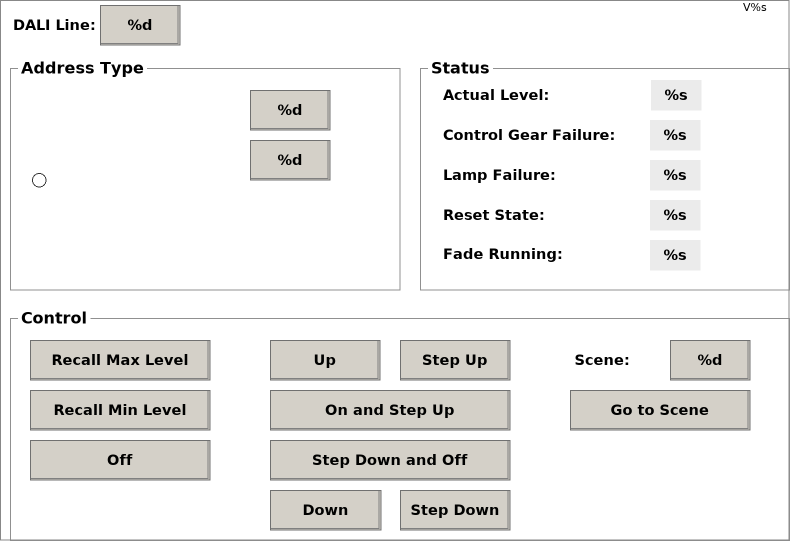
VISUALIZATION Visu_Part102Commands  // 790x541
    GroupBox (10,310 780x231), "Control"
        Button (20,130 180x40), "Off"
            OnMouseClick: execute { DALI_Commissioning.fbPart102Commands.bOff := TRUE; }
        Button (20,80 180x40), "Recall Min Level"
            OnMouseClick: execute { DALI_Commissioning.fbPart102Commands.bRecallMinLevel := TRUE; }
        Button (20,30 180x40), "Recall Max Level"
            OnMouseClick: execute { DALI_Commissioning.fbPart102Commands.bRecallMaxLevel := TRUE; }
        Button (260,180 111x40), "Down"
            OnMouseClick: execute { DALI_Commissioning.fbPart102Commands.bDown := TRUE; }
        Button (390,180 110x40), "Step Down"
            OnMouseClick: execute { DALI_Commissioning.fbPart102Commands.bStepDown := TRUE; }
        Button (260,130 240x40), "Step Down and Off"
            OnMouseClick: execute { DALI_Commissioning.fbPart102Commands.bStepDownAndOff := TRUE; }
        Button (660,30 80x40), "%d", text variable: DALI_Commissioning.fbPart102Commands.nScene
            OnMouseClick: write the text variable via Default, min 0, max 15, title "Insert scene number"
        Textfield (550,35 85x30), "Scene:"
        Button (560,80 180x40), "Go to Scene"
            OnMouseClick: execute { DALI_Commissioning.fbPart102Commands.bGotoScene := TRUE; }
        Button (260,80 240x40), "On and Step Up"
            OnMouseClick: execute { DALI_Commissioning.fbPart102Commands.bOnAndStepUp := TRUE; }
        Button (260,30 110x40), "Up"
            OnMouseClick: execute { DALI_Commissioning.fbPart102Commands.bUp := TRUE; }
        Button (390,30 110x40), "Step Up"
            OnMouseClick: execute { DALI_Commissioning.fbPart102Commands.bStepUp := TRUE; }
    GroupBox (420,60 370x230), "Status"
        Textfield (20,20 200x30), "Actual Level:"
        Textfield (20,60 200x30), "Control Gear Failure:"
        Textfield (231,20 50x30), "%s", text variable: DALI_Commissioning.fbPart102Commands.sActualLevel
        Textfield (230,60 50x30), "%s", text variable: DALI_Commissioning.fbPart102Commands.sControlGearFailure
        Textfield (20,100 200x30), "Lamp Failure:"
        Textfield (230,100 50x30), "%s", text variable: DALI_Commissioning.fbPart102Commands.sLampFailure
        Textfield (20,140 200x30), "Reset State:"
        Textfield (230,140 50x30), "%s", text variable: DALI_Commissioning.fbPart102Commands.sResetState
        Textfield (20,180 200x28), "Fade Running:"
        Textfield (230,180 50x30), "%s", text variable: DALI_Commissioning.fbPart102Commands.sFadeRunning
    GroupBox (10,60 390x230), "Address Type"
        Button (240,30 80x40), "%d", text variable: DALI_Commissioning.fbPart102Commands.nShortAddress
            OnMouseClick: write the text variable via Default, min 0, max 63, title "Insert Short Address"
            OnMouseClick: execute {  }
        RadioButton (20,20 190x200), variable: DALI_Commissioning.fbPart102Commands.eAddressType
            Areas[0]: Text=Short Address
            Areas[1]: Text=Group Address
            Areas[2]: Text=Broadcast
            Areas[3]: Text=Unaddressed
        Button (240,80 80x40), "%d", text variable: DALI_Commissioning.fbPart102Commands.nGroupAddress
            OnMouseClick: write the text variable via Default, min 0, max 15, title "Insert Group Address"
    Rectangle (720,0 70x15), "V%s", text variable: stLibVersion_Tc3_DALI_PLC_Commissioning_Tool.sVersion
    Group (10,5 170x40)
        Textfield (0,0 110x40), "DALI Line:"
        Button (90,0 80x40), "%d", text variable: GVL_Internal.nDALILine
            OnMouseClick: write the text variable via Default, min 1, max 10, title "Choose line"
END_VISUALIZATION

// ---- POUs/DALI/DALI_Setup/VISUs/Visu_DALICommissioning/Visu_Part102SetFading.TcVIS
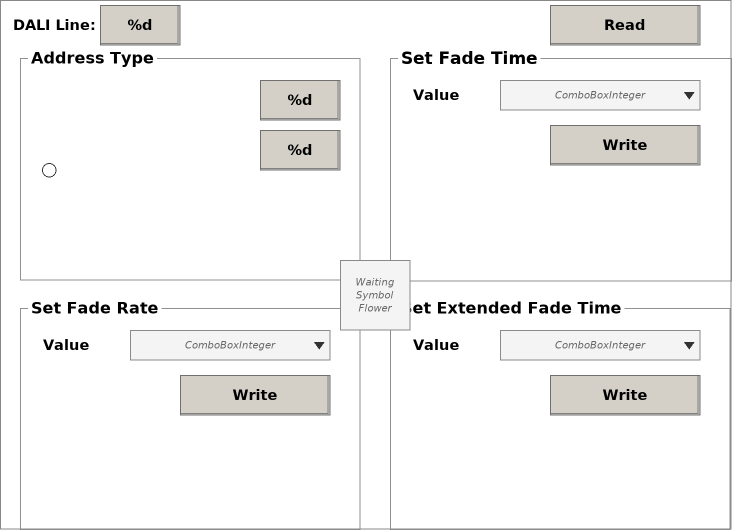
VISUALIZATION Visu_Part102SetFading  // 732x530
    GroupBox (390,50 342x231), "Set Fade Time"
        Textfield (20,30 100x30), "Value"
        ComboBoxInteger (110,30 200x30), variable: DALI_Commissioning.fbPart102SetFading.eFadeTime, text list: 'FadeTime'
        Button (160,75 150x40), "Write"
            OnMouseClick: execute { DALI_Commissioning.fbPart102SetFading.bWriteFadeTime := TRUE; }
    GroupBox (20,50 340x230), "Address Type"
        Button (240,30 80x40), "%d", text variable: DALI_Commissioning.fbPart102SetFading.nShortAddress
            OnMouseClick: write the text variable via Default, min 0, max 63, title "Insert Short Address"
        RadioButton (20,20 190x200), variable: DALI_Commissioning.fbPart102SetFading.eAddressType
            Areas[0]: Text=Short Address
            Areas[1]: Text=Group Address
            Areas[2]: Text=Broadcast
            Areas[3]: Text=Unaddressed
        Button (240,80 80x40), "%d", text variable: DALI_Commissioning.fbPart102SetFading.nGroupAddress
            OnMouseClick: write the text variable via Default, min 0, max 15, title "Insert Group Address"
    GroupBox (20,300 340x230), "Set Fade Rate"
        Textfield (20,30 100x30), "Value"
        ComboBoxInteger (110,30 200x30), variable: DALI_Commissioning.fbPart102SetFading.eFadeRate, text list: 'FadeRate'
        Button (160,75 150x40), "Write"
            OnMouseClick: execute { DALI_Commissioning.fbPart102setFading.bWriteFadeRate := TRUE; }
    GroupBox (390,300 340x230), "Set Extended Fade Time"
        Textfield (20,30 100x30), "Value"
        ComboBoxInteger (110,30 200x30), tooltip "Extended Fade Time only valid if Fade Time equals 0!", variable: DALI_Commissioning.fbPart102SetFading.eExtendedFadeTime, input disabled if: DALI_Commissioning.fbPart102SetFading.bNoFadeTime, text list: 'ExtendedFadeTime'
        Button (160,75 150x40), "Write", tooltip "Extended Fade Time only valid if Fade Time equals 0!", invisible if: DALI_Commissioning.fbPart102SetFading.bNoFadeTime, input disabled if: DALI_Commissioning.fbPart102SetFading.bNoFadeTime
            OnMouseClick: execute { DALI_Commissioning.fbPart102SetFading.bWriteExtendedFadeTime:=true; }
    Button (550,5 150x40), "Read", tooltip "Reads all Fading Parameters", invisible if: ( DALI_Commissioning.fbPart102SetFading.eAddressType >=1), input disabled if: ( DALI_Commissioning.fbPart102SetFading.eAddressType >=1)
        OnMouseClick: execute { DALI_Commissioning.fbPart102SetFading.bRead := TRUE; }
    WaitingSymbolFlower (340,260 70x70), invisible if: DALI_Commissioning.fbPart102SetFading.bHideWaitSymbol
    Group (10,5 170x40)
        Textfield (0,0 110x40), "DALI Line:"
        Button (90,0 80x40), "%d", text variable: GVL_Internal.nDALILine
            OnMouseClick: write the text variable via Default, min 1, max 10, title "Choose line"
END_VISUALIZATION
